(* IEC 61131-3 sources: Industry-PLC-LLM/data/PLCBEAD_repo/PLCBEAD_PLCEmbed-main/PLC-BEAD/Source/GEB/C_TO_K, 1 file *)

(* ---- C_TO_K.ST ---- *)
FUNCTION C_TO_K:REAL
	VAR_INPUT
		CELSIUS :	REAL;
	END_VAR

	C_TO_K := CELSIUS - 273.15;
END_FUNCTION

PROGRAM program0
  VAR
    LocalVar0 : REAL;
    CEIL5_OUT : REAL;
  END_VAR

  CEIL5_OUT := C_TO_K(LocalVar0);
END_PROGRAM
